Fanuc KAREL source: compact_preamble.KL

PROGRAM KB00151
%NOLOCKGROUP
VAR
P1 : STRING[80];P2 : ARRAY[4] OF STRING[80];P3:INTEGER;P4:INTEGER
BEGIN
P1='A'
P3=1
P4=1
RMCN_SEND(P1,P2,P3,P4)
END KB00151
